(* PLC project Blank Project, HUST test 1.0, author wxy *)
(* stored: creationDateTime 2017-01-14T19:11:40, version 1.0, modificationDateTime 2021-01-12T11:11:24 *)

FUNCTION_BLOCK PPIInfo
  VAR
    CURPOS : Axis_Info;
  END_VAR
  VAR_INPUT
    Axis : INT;
  END_VAR
  VAR
    itpc : LREAL;
    itp : LREAL;
    itvc : LREAL;
    itv : LREAL;
    ita : LREAL;
    ppc : UDINT;
    INTERP : Axis_Info;
    INTERPC : Axis_Info;
    INTERV : Axis_Info;
    INTERVC : Axis_Info;
    INTERDP : Axis_Info;
    P0POS : Axis_Info;
    p0p : UDINT;
    PCC : Axis_Info;
    pc : LREAL;
    STATE : Axis_Info;
    MPP : Axis_Info;
    VMAX : Axis_Info;
    AMAX : Axis_Info;
    JMAX : Axis_Info;
    LMTL : Axis_Info;
    AMOD : Axis_Info;
    ERRORID : Axis_Info;
    ABORTFLAG : Axis_Info;
    LMTH : Axis_Info;
    Block1 : Axis_Info;
    qw : QTOUCH_WRITE;
  END_VAR
  VAR  (* added by the conversion: wires and edge detectors of the diagram *)
    _UDINT_TO_INT55_OUT : INT;
    _UDINT_TO_INT87_OUT : INT;
    _UDINT_TO_INT73_OUT : INT;
    _UDINT_TO_INT25_OUT : INT;
    _UDINT_TO_INT35_OUT : INT;
    _LREAL_TO_INT61_OUT : INT;
    _LREAL_TO_INT54_OUT : INT;
    _LREAL_TO_INT38_OUT : INT;
    _LREAL_TO_INT60_OUT : INT;
    _LREAL_TO_INT45_OUT : INT;
    _LREAL_TO_INT70_OUT : INT;
    _LREAL_TO_INT42_OUT : INT;
    _LREAL_TO_INT77_OUT : INT;
    _LREAL_TO_INT92_OUT : INT;
    _LREAL_TO_INT43_OUT : INT;
    _LREAL_TO_INT44_OUT : INT;
    _LREAL_TO_INT82_OUT : INT;
    _LREAL_TO_INT49_OUT : INT;
    _BOOL_TO_UDINT97_OUT : UDINT;
  END_VAR

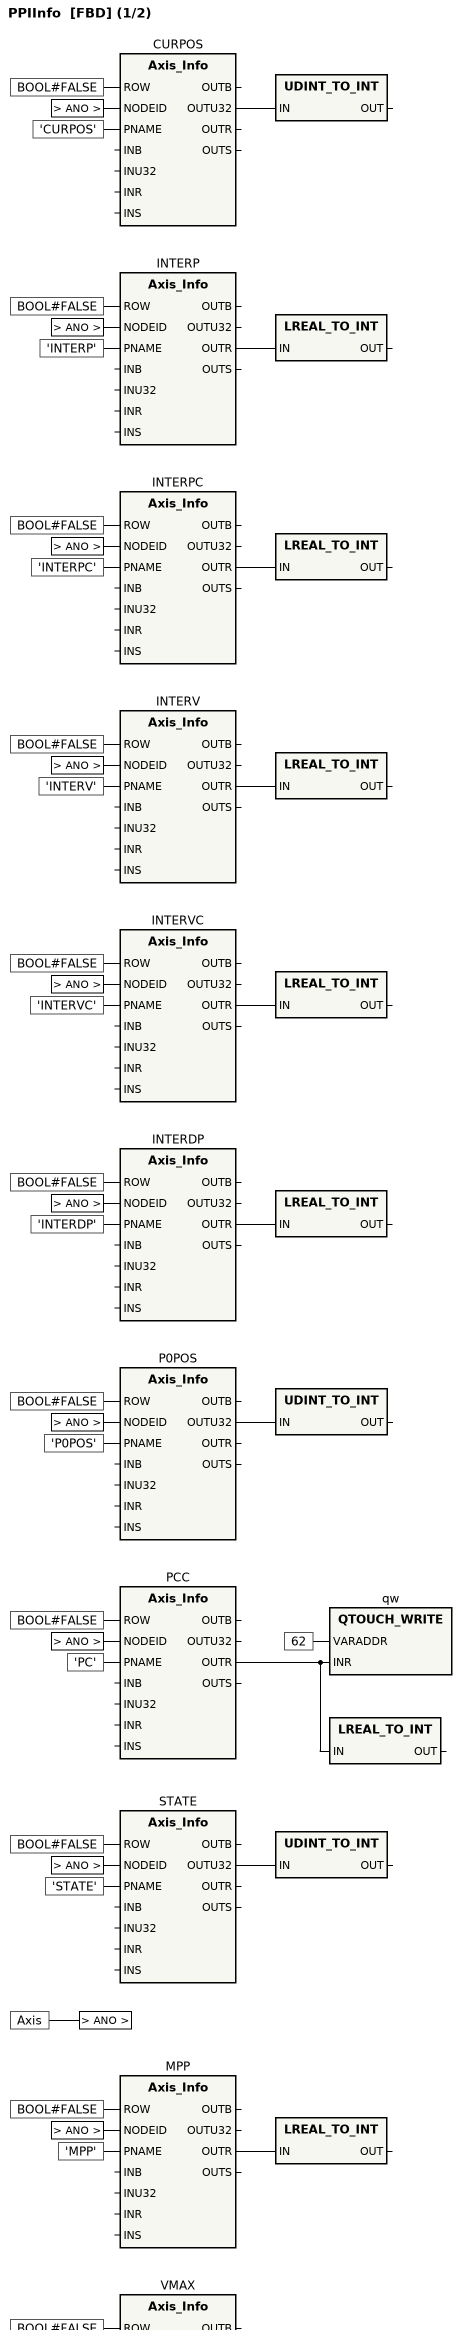
(* FBD diagram, written out as Structured Text *)
STATE(ROW := BOOL#FALSE, NODEID := Axis, PNAME := 'STATE');
ERRORID(ROW := BOOL#FALSE, NODEID := Axis, PNAME := 'ERRORID');
_UDINT_TO_INT55_OUT := UDINT_TO_INT(STATE.OUTU32);
_UDINT_TO_INT87_OUT := UDINT_TO_INT(ERRORID.OUTU32);
ABORTFLAG(ROW := BOOL#FALSE, NODEID := Axis, PNAME := 'ABORTFLAG');
_UDINT_TO_INT73_OUT := UDINT_TO_INT(ABORTFLAG.OUTU32);
CURPOS(ROW := BOOL#FALSE, NODEID := Axis, PNAME := 'CURPOS');
_UDINT_TO_INT25_OUT := UDINT_TO_INT(CURPOS.OUTU32);
P0POS(ROW := BOOL#FALSE, NODEID := Axis, PNAME := 'P0POS');
_UDINT_TO_INT35_OUT := UDINT_TO_INT(P0POS.OUTU32);
INTERP(ROW := BOOL#FALSE, NODEID := Axis, PNAME := 'INTERP');
VMAX(ROW := BOOL#FALSE, NODEID := Axis, PNAME := 'VMAX');
_LREAL_TO_INT61_OUT := LREAL_TO_INT(INTERP.OUTR);
_LREAL_TO_INT54_OUT := LREAL_TO_INT(VMAX.OUTR);
INTERPC(ROW := BOOL#FALSE, NODEID := Axis, PNAME := 'INTERPC');
AMAX(ROW := BOOL#FALSE, NODEID := Axis, PNAME := 'AMAX');
_LREAL_TO_INT38_OUT := LREAL_TO_INT(INTERPC.OUTR);
_LREAL_TO_INT60_OUT := LREAL_TO_INT(AMAX.OUTR);
PCC(ROW := BOOL#FALSE, NODEID := Axis, PNAME := 'PC');
qw(VARADDR := 62, INR := PCC.OUTR);
_LREAL_TO_INT45_OUT := LREAL_TO_INT(PCC.OUTR);
JMAX(ROW := BOOL#FALSE, NODEID := Axis, PNAME := 'JMAX');
_LREAL_TO_INT70_OUT := LREAL_TO_INT(JMAX.OUTR);
INTERV(ROW := BOOL#FALSE, NODEID := Axis, PNAME := 'INTERV');
LMTL(ROW := BOOL#FALSE, NODEID := Axis, PNAME := 'LMTL');
_LREAL_TO_INT42_OUT := LREAL_TO_INT(INTERV.OUTR);
_LREAL_TO_INT77_OUT := LREAL_TO_INT(LMTL.OUTR);
LMTH(ROW := BOOL#FALSE, NODEID := Axis, PNAME := 'LMTH');
_LREAL_TO_INT92_OUT := LREAL_TO_INT(LMTH.OUTR);
INTERVC(ROW := BOOL#FALSE, NODEID := Axis, PNAME := 'INTERVC');
_LREAL_TO_INT43_OUT := LREAL_TO_INT(INTERVC.OUTR);
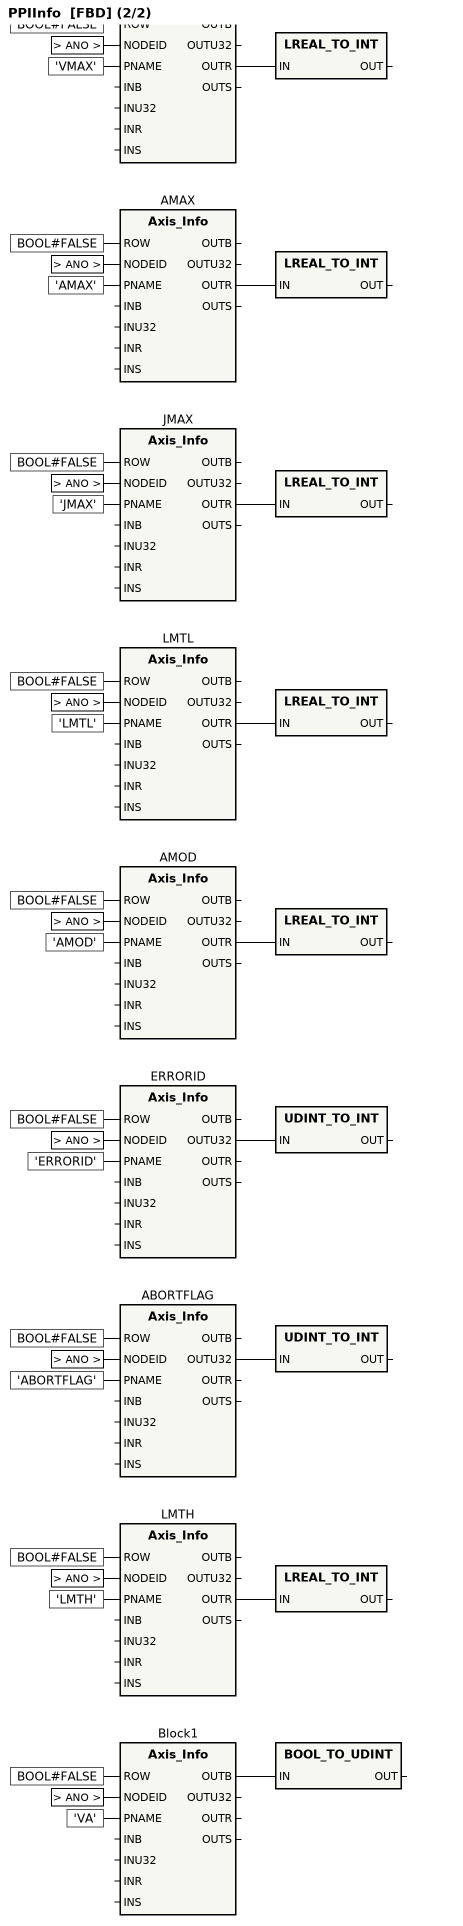
INTERDP(ROW := BOOL#FALSE, NODEID := Axis, PNAME := 'INTERDP');
AMOD(ROW := BOOL#FALSE, NODEID := Axis, PNAME := 'AMOD');
_LREAL_TO_INT44_OUT := LREAL_TO_INT(INTERDP.OUTR);
_LREAL_TO_INT82_OUT := LREAL_TO_INT(AMOD.OUTR);
MPP(ROW := BOOL#FALSE, NODEID := Axis, PNAME := 'MPP');
_LREAL_TO_INT49_OUT := LREAL_TO_INT(MPP.OUTR);
Block1(ROW := BOOL#FALSE, NODEID := Axis, PNAME := 'VA');
_BOOL_TO_UDINT97_OUT := BOOL_TO_UDINT(Block1.OUTB);
END_FUNCTION_BLOCK

FUNCTION_BLOCK vtst
  VAR_INPUT
    us : USINT;
    ui : UINT;
    i16 : INT;
    ud : UDINT;
    ul : ULINT;
    i32 : DINT;
    i64 : LINT;
    r32 : REAL;
    r64 : LREAL;
  END_VAR
  VAR
    ttt : INT;
  END_VAR

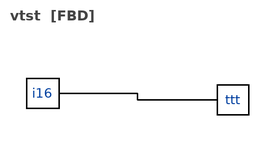
(* FBD diagram, written out as Structured Text *)
ttt := i16;
END_FUNCTION_BLOCK

FUNCTION_BLOCK InitServo
  VAR_INPUT
    AxisID : INT;
    targetMode : USINT;
  END_VAR
  VAR
    Block1 : TON;
    Block3 : TON;
    mi : MC_Init;
    mp : MC_Power;
    ssc : SVRO_CONTROL;
    mmr : MC_Reset;
    jjk : U16_B16;
    pp12 : PPIInfo;
    iir : IP_READ2;
    kkl : B16_U16;
    BGN : BOOL;
  END_VAR
  VAR_OUTPUT
    InitDone : BOOL;
  END_VAR
  VAR
    MCSetP : MC_SetPosition;
    rtii : R_TRIG;
    AXIS_MODE : SVRO_MODE;
    Axis_ActMode : USINT;
  END_VAR

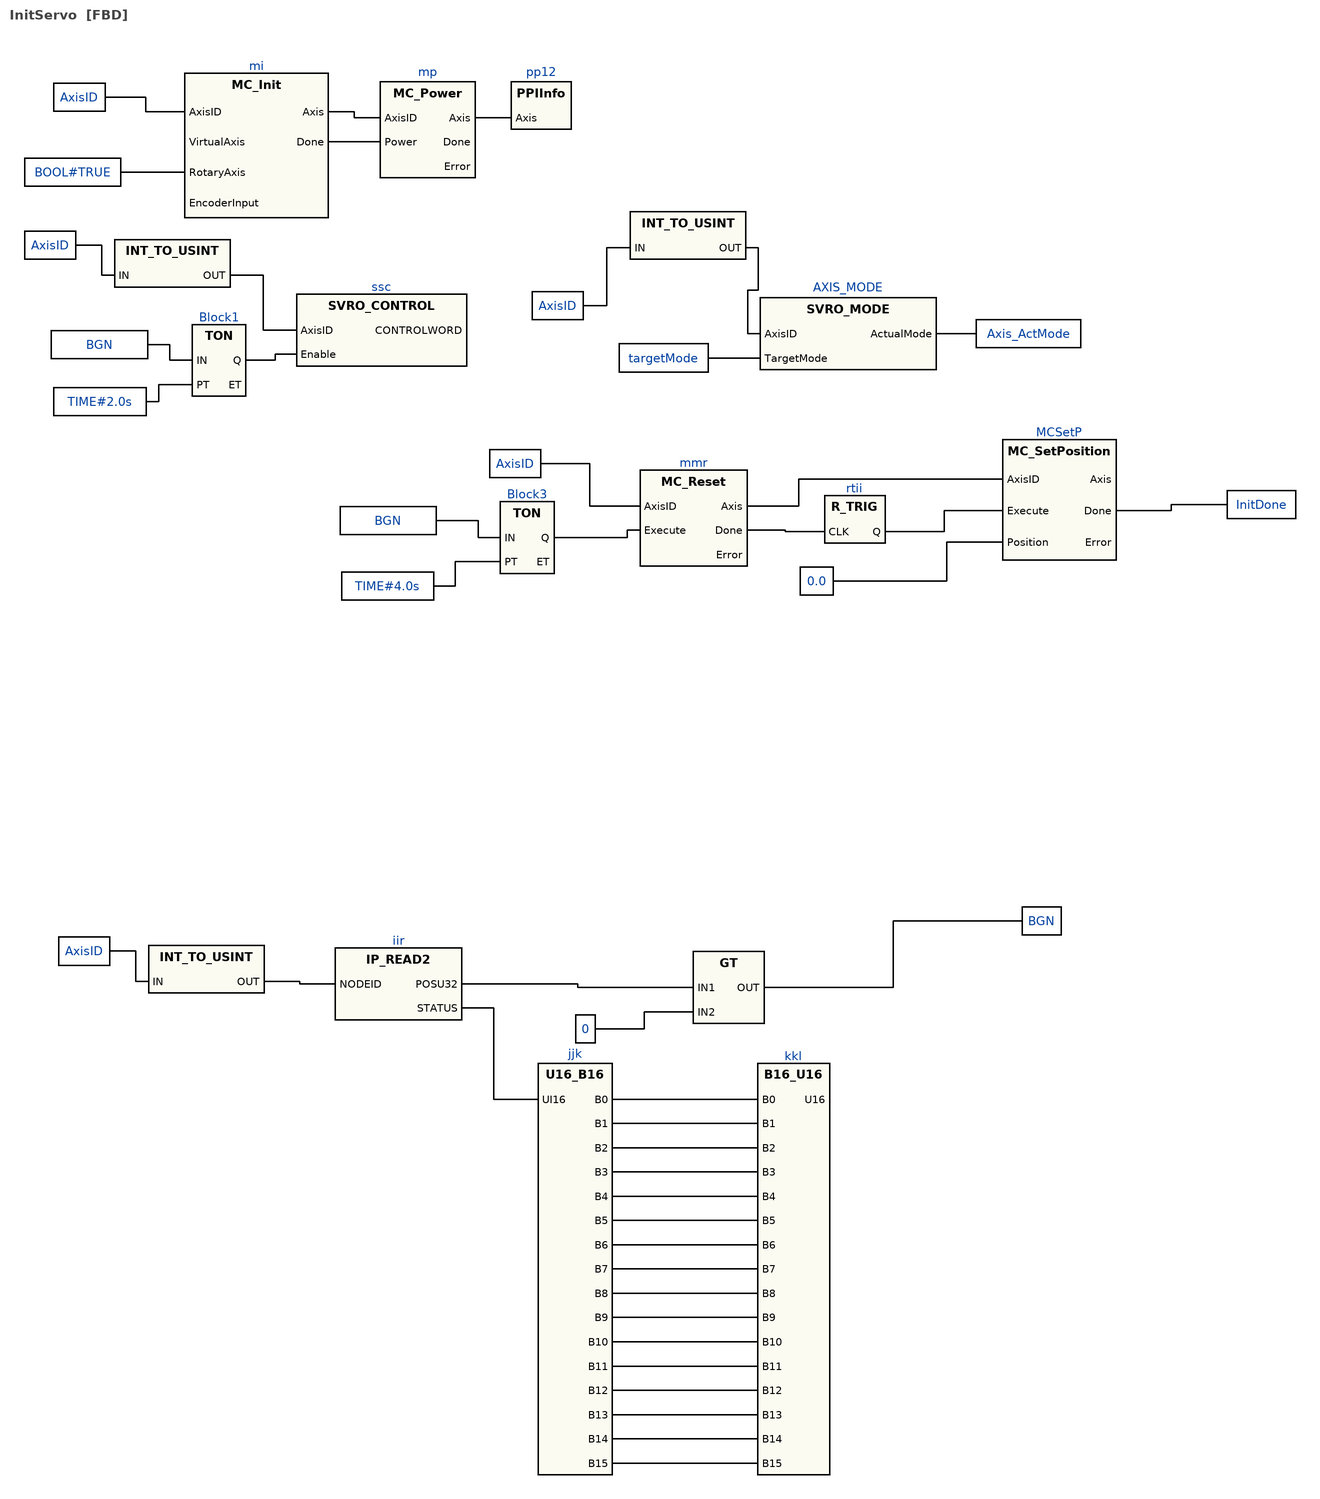
(* FBD diagram, written out as Structured Text *)
AXIS_MODE(AxisID := INT_TO_USINT(AxisID), TargetMode := targetMode);
Axis_ActMode := AXIS_MODE.ActualMode;
Block3(IN := BGN, PT := TIME#4.0s);
mmr(AxisID := AxisID, Execute := Block3.Q);
rtii(CLK := mmr.Done);
MCSetP(AxisID := mmr.Axis, Execute := rtii.Q, Position := 0.0);
InitDone := MCSetP.Done;
iir(NODEID := INT_TO_USINT(AxisID));
BGN := iir.POSU32 > 0;
mi(AxisID := AxisID, RotaryAxis := BOOL#TRUE);
mp(AxisID := mi.Axis, Power := mi.Done);
pp12(Axis := mp.Axis);
Block1(IN := BGN, PT := TIME#2.0s);
ssc(AxisID := INT_TO_USINT(AxisID), Enable := Block1.Q);
jjk(UI16 := iir.STATUS);
kkl(B0 := jjk.B0, B1 := jjk.B1, B2 := jjk.B2, B3 := jjk.B3, B4 := jjk.B4, B5 := jjk.B5, B6 := jjk.B6, B7 := jjk.B7, B8 := jjk.B8, B9 := jjk.B9, B10 := jjk.B10, B11 := jjk.B11, B12 := jjk.B12, B13 := jjk.B13, B14 := jjk.B14, B15 := jjk.B15);
END_FUNCTION_BLOCK

FUNCTION_BLOCK Axis_Mode1
  VAR_INPUT
    En_in : BOOL;
    stop_in : BOOL;
    Axis_No : INT;
    dis_in : LREAL;
    vel_max : LREAL;
  END_VAR
  VAR
    decelerate : BOOL := 0;
    Vel_in : LREAL := 8.0;
  END_VAR
  VAR_INPUT
    acc_in : LREAL;
  END_VAR
  VAR
    T1 : TON;
    t1_up : BOOL;
    T2 : TON;
    t2_up : BOOL;
    T3 : TON;
    t3_up : BOOL;
    T4 : TON;
    t4_up : BOOL;
    L1 : BOOL;
    L2 : BOOL;
    L3 : BOOL;
    L4 : BOOL;
    L5 : BOOL;
    L6 : INT;
    done_1 : BOOL;
    done_2 : BOOL;
    rela1 : MC_Relative;
    rela2 : MC_Relative;
    rela3 : MC_Relative;
    rela4 : MC_Relative;
    rela5 : MC_Relative;
    rela6 : MC_Relative;
    rela7 : MC_Relative;
    rela8 : MC_Relative;
    HALT1 : MC_Halt;
    HALT2 : MC_Halt;
    HALT3 : MC_Halt;
    HALT4 : MC_Halt;
    HALT5 : MC_Halt;
    HALT6 : MC_Halt;
    HALT7 : MC_Halt;
    HALT8 : MC_Halt;
  END_VAR

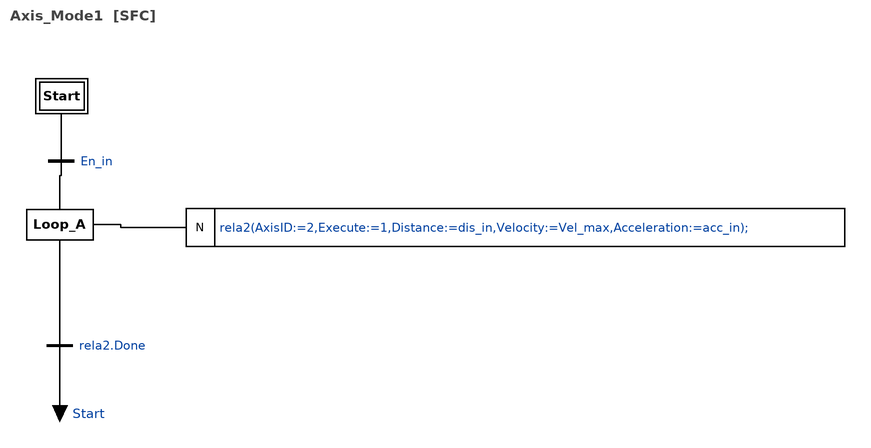
INITIAL_STEP Start:
END_STEP
TRANSITION FROM Start TO Loop_A
  := En_in;
END_TRANSITION
STEP Loop_A:
  LOOP_A_INLINE1(N);
END_STEP
ACTION LOOP_A_INLINE1:
  rela2(AxisID:=2,Execute:=1,Distance:=dis_in,Velocity:=Vel_max,Acceleration:=acc_in);
END_ACTION
TRANSITION FROM Loop_A TO Start
  := rela2.Done;
END_TRANSITION
END_FUNCTION_BLOCK

FUNCTION_BLOCK ZERO
  VAR_INPUT
    En_in : BOOL;
    ActPos : LREAL;
  END_VAR
  VAR
    rr : RBUF_READ;
    Backward : BOOL;
    Forward : BOOL;
  END_VAR
  VAR_OUTPUT
    ZeroDone : BOOL;
  END_VAR
  VAR
    MC_Vel : MC_Velocity;
  END_VAR
  VAR_INPUT
    AxisID : INT;
  END_VAR
  VAR
    AA : MC_Absolute;
    Halt : MC_Halt;
  END_VAR

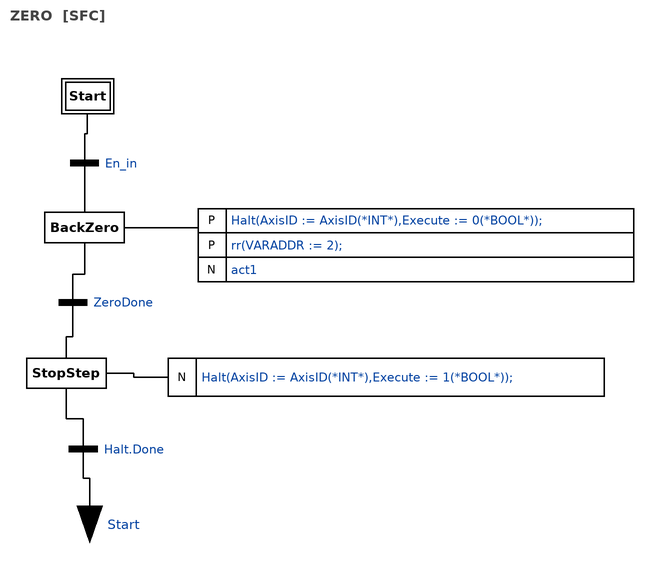
INITIAL_STEP Start:
END_STEP
TRANSITION FROM Start TO BackZero
  := En_in;
END_TRANSITION
STEP BackZero:
  BACKZERO_INLINE1(P);
  BACKZERO_INLINE2(P);
  act1(N);
END_STEP
ACTION BACKZERO_INLINE1:
  Halt(AxisID := AxisID(*INT*),Execute := 0(*BOOL*));
END_ACTION
ACTION BACKZERO_INLINE2:
  rr(VARADDR := 2);
END_ACTION
TRANSITION FROM BackZero TO StopStep
  := ZeroDone;
END_TRANSITION
STEP StopStep:
  STOPSTEP_INLINE3(N);
END_STEP
ACTION STOPSTEP_INLINE3:
  Halt(AxisID := AxisID(*INT*),Execute := 1(*BOOL*));
END_ACTION
TRANSITION FROM StopStep TO Start
  := Halt.Done;
END_TRANSITION

ACTION act1:
if ActPos - rr.OUTR >500.0 then
  MC_Vel(AxisID := AxisID(*INT*),Execute := 1(*BOOL*),Velocity := -0.1(*LREAL*),Acceleration := 0.1(*LREAL*));
  ZeroDone := 0;
elsif ActPos - rr.OUTR >50.0 and ActPos - rr.OUTR <=500.0 then
  MC_Vel(AxisID := AxisID(*INT*),Execute := 1(*BOOL*),Velocity := -0.01(*LREAL*),Acceleration := 0.1(*LREAL*));
  ZeroDone := 0;
elsif ActPos - rr.OUTR <-500.0 then
  MC_Vel(AxisID := AxisID(*INT*),Execute := 1(*BOOL*),Velocity := 0.1(*LREAL*),Acceleration := 0.1(*LREAL*));
  ZeroDone := 0; 
elsif ActPos - rr.OUTR >=-500.0 and ActPos - rr.OUTR <-50.0 then
  MC_Vel(AxisID := AxisID(*INT*),Execute := 1(*BOOL*),Velocity := 0.01(*LREAL*),Acceleration := 0.1(*LREAL*));
  ZeroDone := 0; 
else
 ZeroDone := 1;
 MC_Vel(AxisID := AxisID(*INT*),Execute := 0(*BOOL*),Velocity := 0(*LREAL*),Acceleration := 0.1(*LREAL*));
end_if;
              
END_ACTION
END_FUNCTION_BLOCK

PROGRAM main_fbd
  VAR
    bServoOn : BOOL := FALSE;
    ctrlWord : UINT;
    DigIn_LWord : UINT;
    DigIn_HWord : UINT;
    DigOut_LWord : UINT := 100;
    DigOut_HWord : UINT := 200;
    bDoRelative : BOOL;
    Axis_ActMode : USINT;
    Axis_ActTorque : INT;
    Axis_ActCurrent : INT;
    AXIS_READ2 : IP_READ2;
    Axis_ActPos : UDINT;
    Axis_ActStatusWd : UINT;
    Axis_ActPos2 : UDINT;
    Axis_PosCmd2 : UDINT;
    Axis_deltaPos : UDINT;
    rss : RS;
    dis : INT;
    acc : INT := 1;
    vel : INT := 1;
    InitAxis2 : InitServo;
    modeSet : USINT := 8;
    torqueSet : INT := 0;
    Axis2_R_Torque : TORQUE_READ;
    Axis2_W_Trq : TORQUE_WRITE;
    ClrErr : SVRO_CLEARFAULT;
    bClearErr : BOOL;
    AXISMODE1 : Axis_Mode1;
    ModeEn : BOOL;
    RT : R_TRIG;
    RT1 : R_TRIG;
    MCZero : ZERO;
    rr : RBUF_READ;
  END_VAR

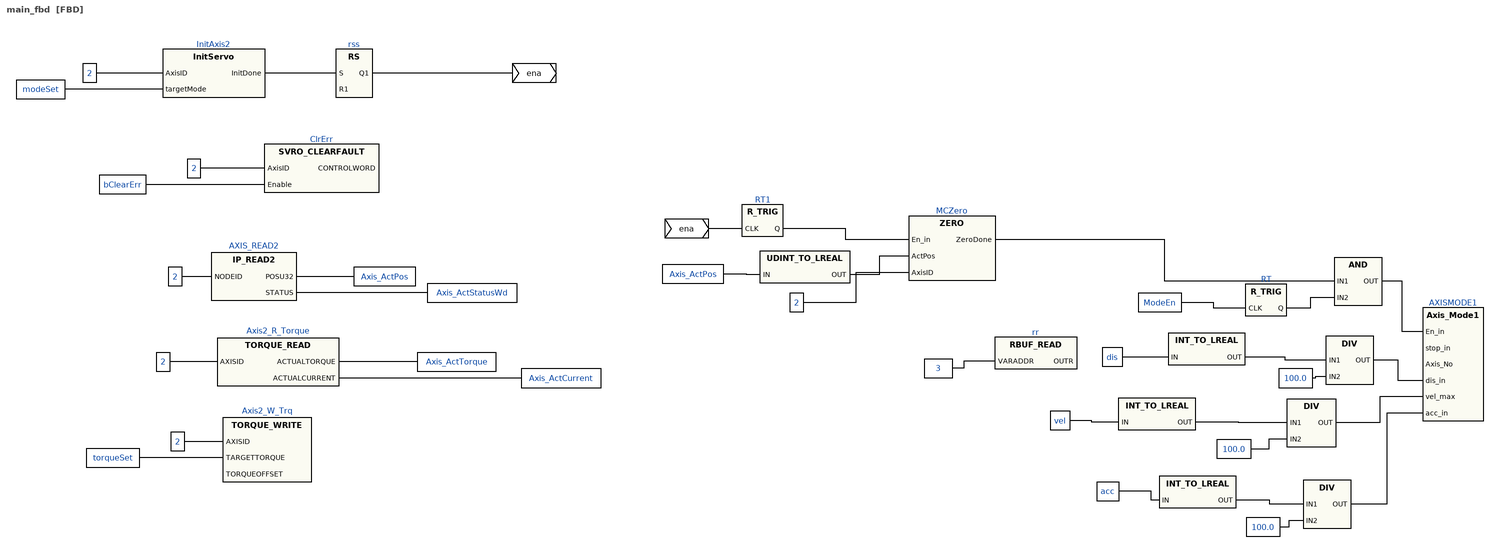
(* FBD diagram, written out as Structured Text *)
AXIS_READ2(NODEID := 2);
Axis_ActPos := AXIS_READ2.POSU32;
Axis_ActStatusWd := AXIS_READ2.STATUS;
Axis2_R_Torque(AXISID := 2);
Axis_ActTorque := Axis2_R_Torque.ACTUALTORQUE;
Axis_ActCurrent := Axis2_R_Torque.ACTUALCURRENT;
InitAxis2(AxisID := 2, targetMode := modeSet);
rss(S := InitAxis2.InitDone);
ClrErr(AxisID := 2, Enable := bClearErr);
RT1(CLK := rss.Q1);
MCZero(En_in := RT1.Q, ActPos := UDINT_TO_LREAL(Axis_ActPos), AxisID := 2);
RT(CLK := ModeEn);
AXISMODE1(En_in := MCZero.ZeroDone AND RT.Q, dis_in := INT_TO_LREAL(dis) / 100.0, vel_max := INT_TO_LREAL(vel) / 100.0, acc_in := INT_TO_LREAL(acc) / 100.0);
rr(VARADDR := 3);
Axis2_W_Trq(AXISID := 2, TARGETTORQUE := torqueSet);
END_PROGRAM

CONFIGURATION conf
  RESOURCE src ON PLC
    TASK tsk(INTERVAL := T#4ms, PRIORITY := 0);
    PROGRAM ref : main_fbd;
  END_RESOURCE
END_CONFIGURATION
